// TIA Portal V17 export
// export: Created 2023-12-05T13:40:23.1396888Z, ExportSetting WithDefaults, DisplayName Totally Integrated Automation Portal, DisplayVersion V17, DisplayName TIA Portal Openness, DisplayVersion V17, DisplayName TIA Portal Version Control Interface, DisplayVersion V17, DisplayName SINAMICS Startdrive Advanced, DisplayVersion V17, DisplayName SINAMICS Startdrive G130, G150, S120, S150, SINAMICS MV, S210, DisplayVersion V17, DisplayName SINAMICS Startdrive G110M, G120, G120C, G120D, G120P, G115D, DisplayVersion V17, DisplayName STEP 7 Professional, DisplayVersion V17, DisplayName STEP 7 Safety, DisplayVersion V17, DisplayName WinCC Professional, DisplayVersion V17
FUNCTION "FC533 NPW_V5_1_7 Alarms" : Void   // FC533, LAD
{ S7_Optimized_Access := 'FALSE' }
VERSION : 0.1
// LG 29.06.2022 =>  Changed both blocks (NPWBC 5.1.6 and NPWSC 5.1.6) to new block NPW 5.1.7
// RB 08.09.2021 => Changed name of the block (structures are the same like in STD Block V 5_1_0)
// LM 4.06.2020 => Check for SB V5_1_0
// RB 8.05.2020 => Edited to copy whole alarms on their  IDB addresses
// stored: AutoNumber false, IsIECCheckEnabled false, SetENOAutomatically false, UDAEnableTagReadback false
   VAR_INPUT
      AckStep : Bool;
      "SB DB" : Int;
      "Alarm DB" : Int;
      "Alarm Offset" : Int;
   END_VAR
   VAR_TEMP
      "SB DBW" : Word;
      "AL DBW" : Word;
   END_VAR
BEGIN

NETWORK
TITLE = Initialization
      L     #"SB DB";
      T     #"SB DBW";
      L     #"Alarm DB";
      T     #"AL DBW";
      L     #"Alarm Offset";
      SLD   3;
      LAR1;

NETWORK
TITLE = 
      CLR;
      OPN   DB [#"SB DBW"];
      L     %DBW156;
      OPN   DB [#"AL DBW"];
      T     DBW [AR1, P#0.0];

      OPN   DB [#"SB DBW"];
      A     %DBX167.1;
      OPN   DB [#"AL DBW"];
      =     DBX [AR1, P#11.1];

      OPN   DB [#"SB DBW"];
      A     %DBX174.0;
      OPN   DB [#"AL DBW"];
      =     DBX [AR1, P#17.0];

      OPN   DB [#"SB DBW"];
      A     %DBX174.1;
      OPN   DB [#"AL DBW"];
      =     DBX [AR1, P#17.1];

      OPN   DB [#"SB DBW"];
      A     %DBX174.2;
      OPN   DB [#"AL DBW"];
      =     DBX [AR1, P#17.2];

      OPN   DB [#"SB DBW"];
      A     %DBX174.6;
      OPN   DB [#"AL DBW"];
      =     DBX [AR1, P#17.6];

      OPN   DB [#"SB DBW"];
      A     %DBX174.7;
      OPN   DB [#"AL DBW"];
      =     DBX [AR1, P#17.7];



NETWORK
TITLE = 
      A     #AckStep;
      JCN   eno;
      OPN   DB [#"SB DBW"];
      L     %DBW164;
      OPN   DB [#"AL DBW"];
      T     DBW [AR1, P#8.0];

      OPN   DB [#"SB DBW"];
      L     %DBW166;
      OPN   DB [#"AL DBW"];
      T     DBW [AR1, P#10.0];

      OPN   DB [#"SB DBW"];
      L     %DBW168;
      OPN   DB [#"AL DBW"];
      T     DBW [AR1, P#12.0];

      OPN   DB [#"SB DBW"];
      L     %DBW170;
      OPN   DB [#"AL DBW"];
      T     DBW [AR1, P#14.0];

      OPN   DB [#"SB DBW"];
      A     %DBX175.1;
      OPN   DB [#"AL DBW"];
      =     DBX [AR1, P#18.1];

      OPN   DB [#"SB DBW"];
      A     %DBX175.2;
      OPN   DB [#"AL DBW"];
      =     DBX [AR1, P#18.2];

      OPN   DB [#"SB DBW"];
      A     %DBX175.3;
      OPN   DB [#"AL DBW"];
      =     DBX [AR1, P#18.3];

eno:  NOP   0;
END_FUNCTION
